FUNCTION_BLOCK SimpleNOT (* Simple FB with one algorithm *)
  (* Standard: 61499-1 *)
  (* Version 1.0, 2022-08-30, AK115394 *)
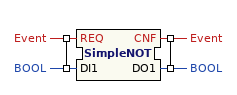
  EVENT_INPUT
    REQ WITH DI1; (* Normal Execution Request *)
  END_EVENT
  EVENT_OUTPUT
    CNF WITH DO1; (* Execution Confirmation *)
  END_EVENT
  VAR_INPUT
    DI1 : BOOL;
  END_VAR
  VAR_OUTPUT
    DO1 : BOOL;
  END_VAR
  ALGORITHM REQ IN ST:
	DO1 := NOT DI1;
  END_ALGORITHM
END_FUNCTION_BLOCK
